// TIA Portal V16 export
// export: Created 2023-08-28T09:37:48.4116382Z, ExportSetting WithDefaults, DisplayName Totally Integrated Automation Portal, DisplayVersion V16 Update 6, DisplayName TIA Portal Version Control Interface, DisplayVersion V16 Update 2, DisplayName TIA Portal Openness, DisplayVersion V16 Update 6, DisplayName STEP 7 Professional, DisplayVersion V16 Update 6, DisplayName STEP 7 Safety, DisplayVersion V16, DisplayName WinCC Advanced, DisplayVersion V16 Update 6
DATA_BLOCK "dbControl of connection Inverters P1"   // DB42
AUTHOR : rtecmer
VERSION : 0.1
// stored: AutoNumber true, DBAccessibleFromOPCUA true, InstanceOfName 06_M_Inverter connection control, InstanceOfType FB
"06_M_Inverter connection control"
   // VAR_INPUT
   //    Is_up_Hz : Bool;
   //    Set_HWork_M : Bool;
   //    setPID_Pompy : Bool;
   //    IsRunInverter_MA : Bool;
   //    IsRunNetwork_MA : Bool;
   //    IsRunInverter_MB : Bool;
   //    IsRunNetwork_MB : Bool;
   //    IsRunNetwork_MC : Bool;
   //    IsRunInverter_MC : Bool;
   //    IsRunNetwork_MD : Bool;
   //    IsRunInverter_MD : Bool;
   //    FC2_Set_50H : Bool;
   //    IsRunInverter1 : Bool;
   //    AlwaysTRUE : Bool;
   //    IsReady_MA : Bool;
   //    IsReady_MB : Bool;
   //    IsReady_MC : Bool;
   //    IsReady_MD : Bool;
   //    IsModeAut : Bool;
   //    FB9_Set_Motor2 : Bool;
   //    FB9_Set_Motor3 : Bool;
   //    FB9_Set_Motor4 : Bool;
   //    IsReady_Inverter : Bool;
   //    ResWorkInverter_to_MaxTime : Bool;
   //    number_pump : Int;
   //    ActivePump : Int;
   // END_VAR
   // VAR_OUTPUT
   //    setSUPV_FM : Bool;
   // END_VAR
   // VAR_IN_OUT
   //    setCMD_FM : Bool;
   //    Timer_OFF_Inverter_M : TOF_TIME;
   //    Timer_Start_Inver_M : TON_TIME;
   //    Timer_Set50Hz_Off_Inver_M : TON_TIME;
   //    Mem_Res_setCMD_MC : Bool;
   // END_VAR
   // VAR
   //    Network_50Hz : Bool;
   // END_VAR
BEGIN
END_DATA_BLOCK
